// TIA Portal V20 export
FUNCTION_BLOCK "Sequence_2_VisionController"   // FB121, LAD
TITLE = Sequence
// Sequence template programmend in ladder logic
// stored: IsIECCheckEnabled true, MemoryReserve 100, Namespace Unit1.Em6, SetENOAutomatically true
   VAR_OUTPUT
      safeState : Bool;
   END_VAR
   VAR
      statSelectedJobNumber { ExternalWritable := 'False'} : DInt;   // Evaluated Job Number
      instSequenceLADControl { ExternalWritable := 'False'} : "LAF_ControlLadSequence";
      instSequenceLADStatus { ExternalWritable := 'False'} : "LAF_StatusLadSequence";
      statResetJobs { ExternalWritable := 'False'} : Bool;
      statPulse { ExternalWritable := 'False'} : Array[0..999] of Bool;
      statTonTimer { ExternalWritable := 'False'} : Array[0..999] of TON_TIME;
   END_VAR
   VAR_TEMP
      tempCustomerAction : Bool;   // Placeholder for possible actions
      tempDo_nothing_and_wait_for_init : Bool;   // Placeholder for doing nothing
      tempSafeStateCondition : Bool;   // Temp Condition for the equipment module to be in a safe state
   END_VAR
   VAR CONSTANT
      STEP_IDLE : DInt := 1;   // Idle Step
      JOB_1_STEP_01 : DInt := 101;   // Template Step
      JOB_1_STEP_11 : DInt := 111;   // Template Step
      JOB_1_STEP_21 : DInt := 121;   // Template Step
      JOB_1_STEP_31 : DInt := 131;   // Template Step
      JOB_1_STEP_91 : DInt := 191;   // Template Step
      JOB_2_STEP_01 : DInt := 201;   // Template Step
      JOB_2_STEP_11 : DInt := 211;   // Template Step
      JOB_2_STEP_21 : DInt := 221;   // Template Step
      JOB_2_STEP_91 : DInt := 291;   // Template Step
      STEP_IMMEDIATE_STOP : DInt := 901;   // Step executed when an immediate stop command is triggered for the sequence (i.e. when unit is in state aborting)
      SeqDelayTime : Time := T#100ms;
      SeqNoDelayTime : Time;
      TRUE : Bool := TRUE;
      FALSE : Bool := FALSE;
   END_VAR
   VAR_TEMP   // added for the SCL form of the ladder/FBD networks
      _w1 : Bool;
   END_VAR
BEGIN

REGION Network 1: BLOCK INFO HEADER
   // (company) / (C) Copyright (year)
   // ---------------------------------------------------------------------------------
   // Title:                             (Title of this block)
   // Comment/Function: (that is implemented in the block)
   // Library/Family:           (that the source is dedicated to)
   // Author:                        (department / person in charge / contact)
   // Target System:          (test system with FW version)
   // Engineering:              TIA Portal (SW version)
   // Restrictions:               (OB types, etc.)
   // Requirements:           (hardware, technological package, etc.)
   // ---------------------------------------------------------------------------------
   // Change log table:
   // Version          | Date             | Signature      | Expert in charge  | Changes applied ------------------------|----------------------|-------------------------|--------------------------------|-----------------------
   // 001.000.000 | yyyy-mm-dd | 0x00000000 | (name of expert) | First released version
END_REGION

REGION Network 2: DESCRIPTION
   // This is a template block provided by the Automation Framework. It can be used to create an own project.
   // The Block Info Header is prepared to put in your own data.
   // Description of the block could be added here and the docu created by Code2Docu.
END_REGION

REGION Network 3: ******************** CONTROL ********************
END_REGION

REGION Network 4: Sequence Control
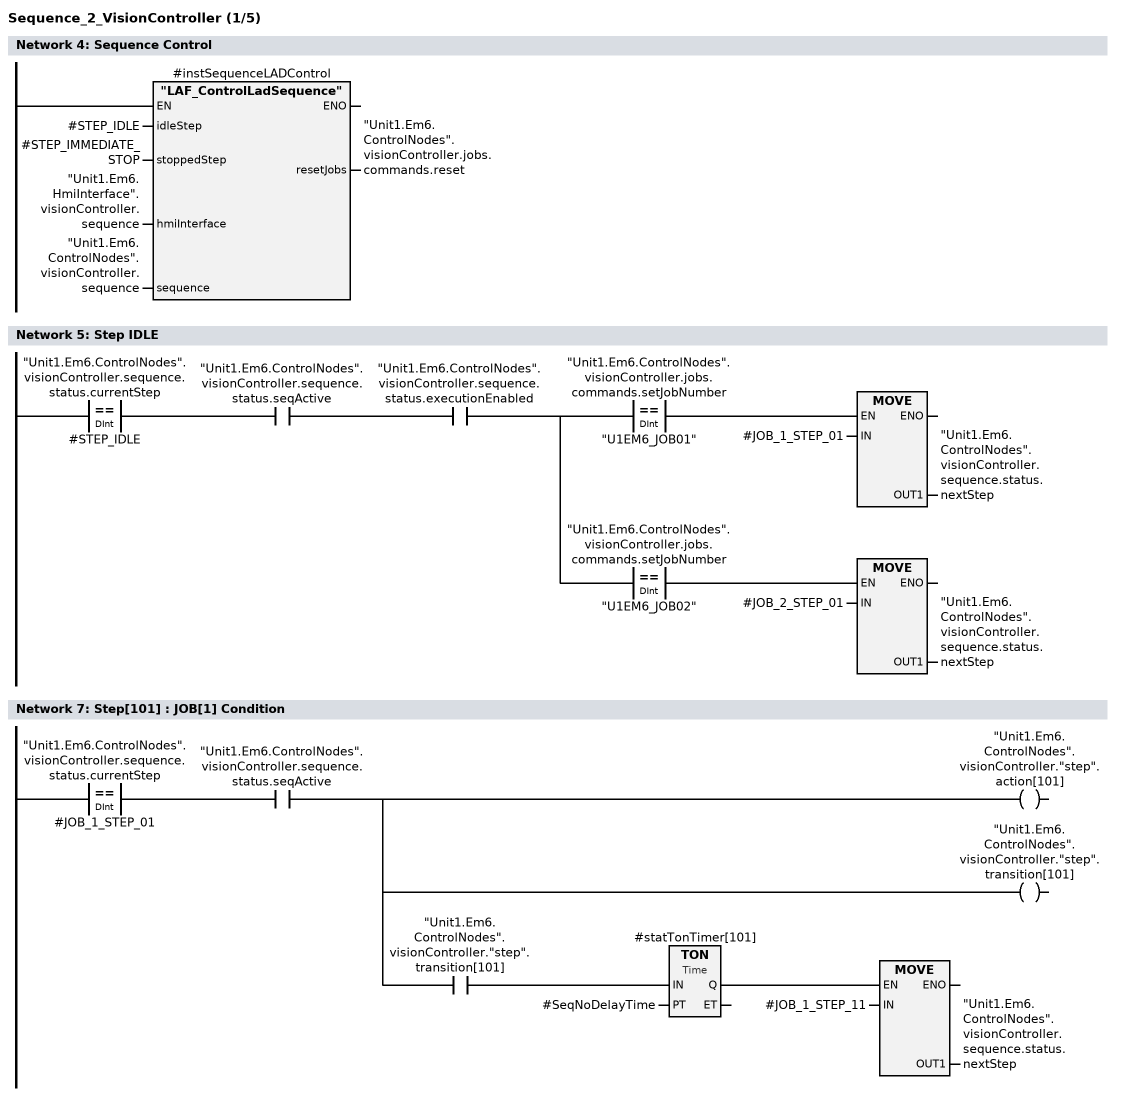
   RUNG wire#powerrail
      #instSequenceLADControl(idleStep := #STEP_IDLE, stoppedStep := #STEP_IMMEDIATE_STOP, hmiInterface := "Unit1.Em6.HmiInterface".visionController.sequence, sequence := "Unit1.Em6.ControlNodes".visionController.sequence, resetJobs => "Unit1.Em6.ControlNodes".visionController.jobs.commands.reset)
   END_RUNG
   // the same network as SCL:
   #instSequenceLADControl(idleStep := #STEP_IDLE,   // "LAF_ControlLadSequence"
                           stoppedStep := #STEP_IMMEDIATE_STOP,
                           hmiInterface := "Unit1.Em6.HmiInterface".visionController.sequence,
                           sequence := "Unit1.Em6.ControlNodes".visionController.sequence,
                           resetJobs => "Unit1.Em6.ControlNodes".visionController.jobs.commands.reset);
END_REGION

REGION Network 5: Step IDLE
   RUNG wire#powerrail
      { S7_Templates := "SrcType := DInt" } EQ_Contact(in1 := "Unit1.Em6.ControlNodes".visionController.sequence.status.currentStep, in2 := #STEP_IDLE)
      Contact( "Unit1.Em6.ControlNodes".visionController.sequence.status.seqActive )
      Contact( "Unit1.Em6.ControlNodes".visionController.sequence.status.executionEnabled )
      wire#w1
      { S7_Templates := "SrcType := DInt" } EQ_Contact(in1 := "Unit1.Em6.ControlNodes".visionController.jobs.commands.setJobNumber, in2 := "U1EM6_JOB01")
      Move(in := #JOB_1_STEP_01, out1 => "Unit1.Em6.ControlNodes".visionController.sequence.status.nextStep)
   END_RUNG
   RUNG wire#w1
      { S7_Templates := "SrcType := DInt" } EQ_Contact(in1 := "Unit1.Em6.ControlNodes".visionController.jobs.commands.setJobNumber, in2 := "U1EM6_JOB02")
      Move(in := #JOB_2_STEP_01, out1 => "Unit1.Em6.ControlNodes".visionController.sequence.status.nextStep)
   END_RUNG
   // the same network as SCL:
   #_w1 := ("Unit1.Em6.ControlNodes".visionController.sequence.status.currentStep = #STEP_IDLE) AND "Unit1.Em6.ControlNodes".visionController.sequence.status.seqActive AND "Unit1.Em6.ControlNodes".visionController.sequence.status.executionEnabled;
   IF #_w1 AND ("Unit1.Em6.ControlNodes".visionController.jobs.commands.setJobNumber = "U1EM6_JOB01") THEN
       "Unit1.Em6.ControlNodes".visionController.sequence.status.nextStep := #JOB_1_STEP_01;
   END_IF;
   IF #_w1 AND ("Unit1.Em6.ControlNodes".visionController.jobs.commands.setJobNumber = "U1EM6_JOB02") THEN
       "Unit1.Em6.ControlNodes".visionController.sequence.status.nextStep := #JOB_2_STEP_01;
   END_IF;
END_REGION

REGION Network 6: ******************** JOB[1] EM INITIALIZED ********************
END_REGION

REGION Network 7: Step[101] : JOB[1] Condition
   RUNG wire#powerrail
      { S7_Templates := "SrcType := DInt" } EQ_Contact(in1 := "Unit1.Em6.ControlNodes".visionController.sequence.status.currentStep, in2 := #JOB_1_STEP_01)
      Contact( "Unit1.Em6.ControlNodes".visionController.sequence.status.seqActive )
      wire#w1
      Coil( "Unit1.Em6.ControlNodes".visionController."step".action[101] )
   END_RUNG
   RUNG wire#w1
      Coil( "Unit1.Em6.ControlNodes".visionController."step".transition[101] )
   END_RUNG
   RUNG wire#w1
      Contact( "Unit1.Em6.ControlNodes".visionController."step".transition[101] )
      { S7_Templates := "time_type := Time" } #statTonTimer[101].TON(pt := #SeqNoDelayTime, et =>)
      Move(in := #JOB_1_STEP_11, out1 => "Unit1.Em6.ControlNodes".visionController.sequence.status.nextStep)
   END_RUNG
   // the same network as SCL:
   "Unit1.Em6.ControlNodes".visionController."step".action[101] := ("Unit1.Em6.ControlNodes".visionController.sequence.status.currentStep = #JOB_1_STEP_01) AND "Unit1.Em6.ControlNodes".visionController.sequence.status.seqActive;
   "Unit1.Em6.ControlNodes".visionController."step".transition[101] := ("Unit1.Em6.ControlNodes".visionController.sequence.status.currentStep = #JOB_1_STEP_01) AND "Unit1.Em6.ControlNodes".visionController.sequence.status.seqActive;
   #statTonTimer[101].TON(IN := ("Unit1.Em6.ControlNodes".visionController.sequence.status.currentStep = #JOB_1_STEP_01) AND "Unit1.Em6.ControlNodes".visionController.sequence.status.seqActive AND "Unit1.Em6.ControlNodes".visionController."step".transition[101],
                          PT := #SeqNoDelayTime);
   IF #statTonTimer[101].Q THEN
       "Unit1.Em6.ControlNodes".visionController.sequence.status.nextStep := #JOB_1_STEP_11;
   END_IF;
END_REGION

REGION Network 8: Step[111] : Vision Controller Ready Check
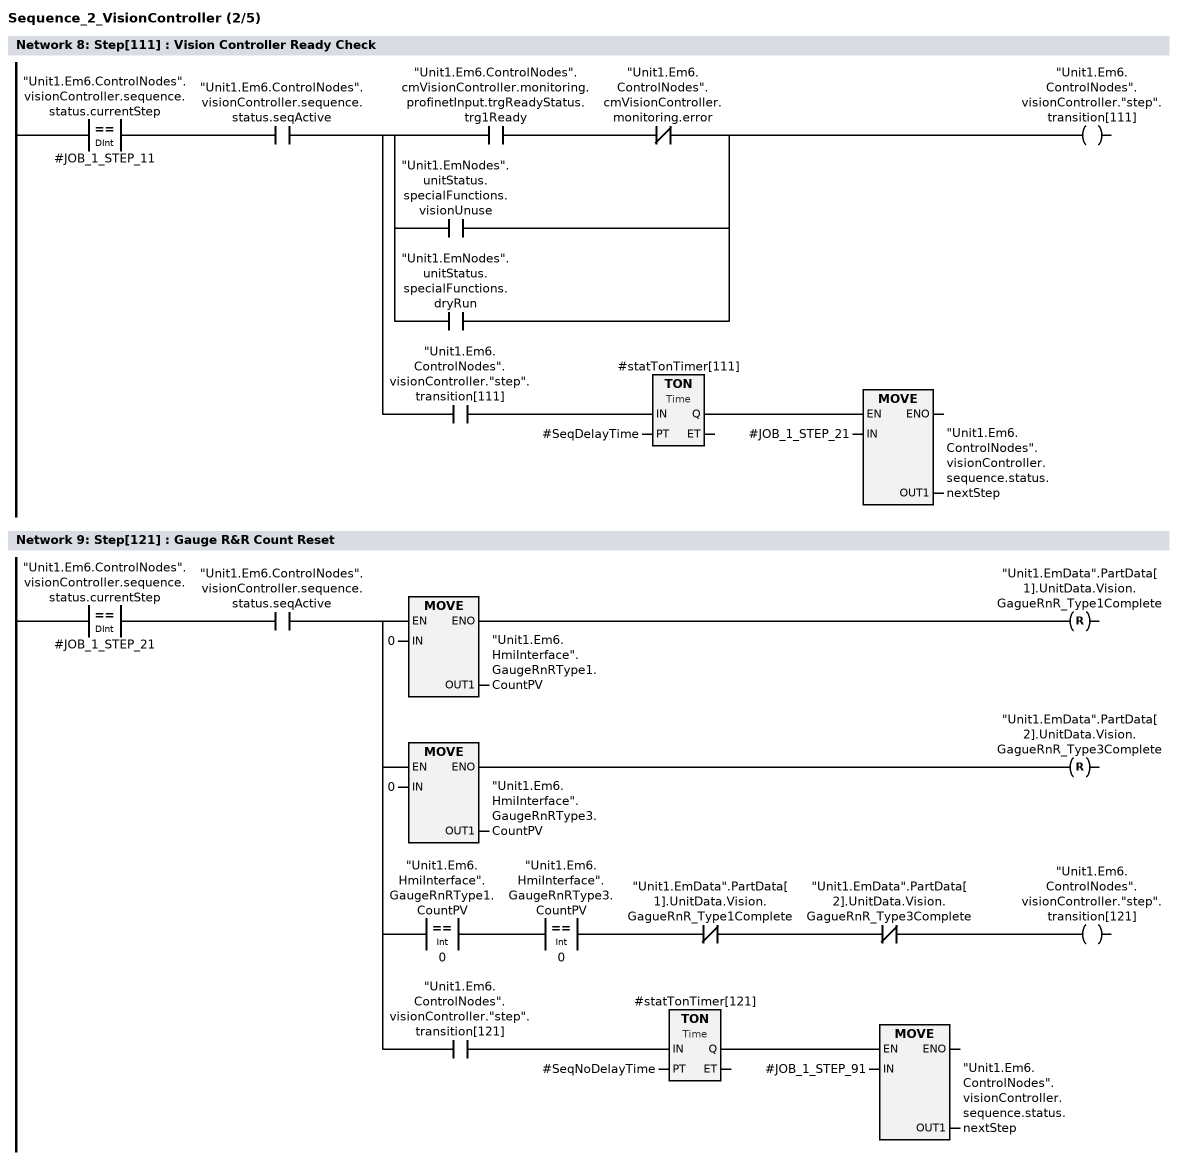
   RUNG wire#powerrail
      { S7_Templates := "SrcType := DInt" } EQ_Contact(in1 := "Unit1.Em6.ControlNodes".visionController.sequence.status.currentStep, in2 := #JOB_1_STEP_11)
      Contact( "Unit1.Em6.ControlNodes".visionController.sequence.status.seqActive )
      wire#w1
      Contact( "Unit1.Em6.ControlNodes".cmVisionController.monitoring.profinetInput.trgReadyStatus.trg1Ready )
      I_Contact( "Unit1.Em6.ControlNodes".cmVisionController.monitoring.error )
      wire#w2
      Coil( "Unit1.Em6.ControlNodes".visionController."step".transition[111] )
   END_RUNG
   RUNG wire#w1
      Contact( "Unit1.EmNodes".unitStatus.specialFunctions.visionUnuse )
   END_RUNG wire#w2
   RUNG wire#w1
      Contact( "Unit1.EmNodes".unitStatus.specialFunctions.dryRun )
   END_RUNG wire#w2
   RUNG wire#w1
      Contact( "Unit1.Em6.ControlNodes".visionController."step".transition[111] )
      { S7_Templates := "time_type := Time" } #statTonTimer[111].TON(pt := #SeqDelayTime, et =>)
      Move(in := #JOB_1_STEP_21, out1 => "Unit1.Em6.ControlNodes".visionController.sequence.status.nextStep)
   END_RUNG
   // the same network as SCL:
   #_w1 := ("Unit1.Em6.ControlNodes".visionController.sequence.status.currentStep = #JOB_1_STEP_11) AND "Unit1.Em6.ControlNodes".visionController.sequence.status.seqActive;
   "Unit1.Em6.ControlNodes".visionController."step".transition[111] := #_w1 AND (("Unit1.Em6.ControlNodes".cmVisionController.monitoring.profinetInput.trgReadyStatus.trg1Ready AND NOT "Unit1.Em6.ControlNodes".cmVisionController.monitoring.error) OR "Unit1.EmNodes".unitStatus.specialFunctions.visionUnuse OR "Unit1.EmNodes".unitStatus.specialFunctions.dryRun);
   #statTonTimer[111].TON(IN := #_w1 AND "Unit1.Em6.ControlNodes".visionController."step".transition[111],
                          PT := #SeqDelayTime);
   IF #statTonTimer[111].Q THEN
       "Unit1.Em6.ControlNodes".visionController.sequence.status.nextStep := #JOB_1_STEP_21;
   END_IF;
END_REGION

REGION Network 9: Step[121] : Gauge R&R Count Reset
   RUNG wire#powerrail
      { S7_Templates := "SrcType := DInt" } EQ_Contact(in1 := "Unit1.Em6.ControlNodes".visionController.sequence.status.currentStep, in2 := #JOB_1_STEP_21)
      Contact( "Unit1.Em6.ControlNodes".visionController.sequence.status.seqActive )
      wire#w1
      Move(in := 0, out1 => "Unit1.Em6.HmiInterface".GaugeRnRType1.CountPV)
      R_Coil( "Unit1.EmData".PartData[1].UnitData.Vision.GagueRnR_Type1Complete )
   END_RUNG
   RUNG wire#w1
      Move(in := 0, out1 => "Unit1.Em6.HmiInterface".GaugeRnRType3.CountPV)
      R_Coil( "Unit1.EmData".PartData[2].UnitData.Vision.GagueRnR_Type3Complete )
   END_RUNG
   RUNG wire#w1
      { S7_Templates := "SrcType := Int" } EQ_Contact(in1 := "Unit1.Em6.HmiInterface".GaugeRnRType1.CountPV, in2 := 0)
      { S7_Templates := "SrcType := Int" } EQ_Contact(in1 := "Unit1.Em6.HmiInterface".GaugeRnRType3.CountPV, in2 := 0)
      I_Contact( "Unit1.EmData".PartData[1].UnitData.Vision.GagueRnR_Type1Complete )
      I_Contact( "Unit1.EmData".PartData[2].UnitData.Vision.GagueRnR_Type3Complete )
      Coil( "Unit1.Em6.ControlNodes".visionController."step".transition[121] )
   END_RUNG
   RUNG wire#w1
      Contact( "Unit1.Em6.ControlNodes".visionController."step".transition[121] )
      { S7_Templates := "time_type := Time" } #statTonTimer[121].TON(pt := #SeqNoDelayTime, et =>)
      Move(in := #JOB_1_STEP_91, out1 => "Unit1.Em6.ControlNodes".visionController.sequence.status.nextStep)
   END_RUNG
   // the same network as SCL:
   #_w1 := ("Unit1.Em6.ControlNodes".visionController.sequence.status.currentStep = #JOB_1_STEP_21) AND "Unit1.Em6.ControlNodes".visionController.sequence.status.seqActive;
   IF #_w1 THEN
       "Unit1.Em6.HmiInterface".GaugeRnRType1.CountPV := 0;
       "Unit1.EmData".PartData[1].UnitData.Vision.GagueRnR_Type1Complete := FALSE;
       "Unit1.Em6.HmiInterface".GaugeRnRType3.CountPV := 0;
       "Unit1.EmData".PartData[2].UnitData.Vision.GagueRnR_Type3Complete := FALSE;
   END_IF;
   "Unit1.Em6.ControlNodes".visionController."step".transition[121] := #_w1 AND ("Unit1.Em6.HmiInterface".GaugeRnRType1.CountPV = 0) AND ("Unit1.Em6.HmiInterface".GaugeRnRType3.CountPV = 0) AND NOT "Unit1.EmData".PartData[1].UnitData.Vision.GagueRnR_Type1Complete AND NOT "Unit1.EmData".PartData[2].UnitData.Vision.GagueRnR_Type3Complete;
   #statTonTimer[121].TON(IN := #_w1 AND "Unit1.Em6.ControlNodes".visionController."step".transition[121],
                          PT := #SeqNoDelayTime);
   IF #statTonTimer[121].Q THEN
       "Unit1.Em6.ControlNodes".visionController.sequence.status.nextStep := #JOB_1_STEP_91;
   END_IF;
END_REGION

REGION Network 10: Step[191] : JOB[1] Step End
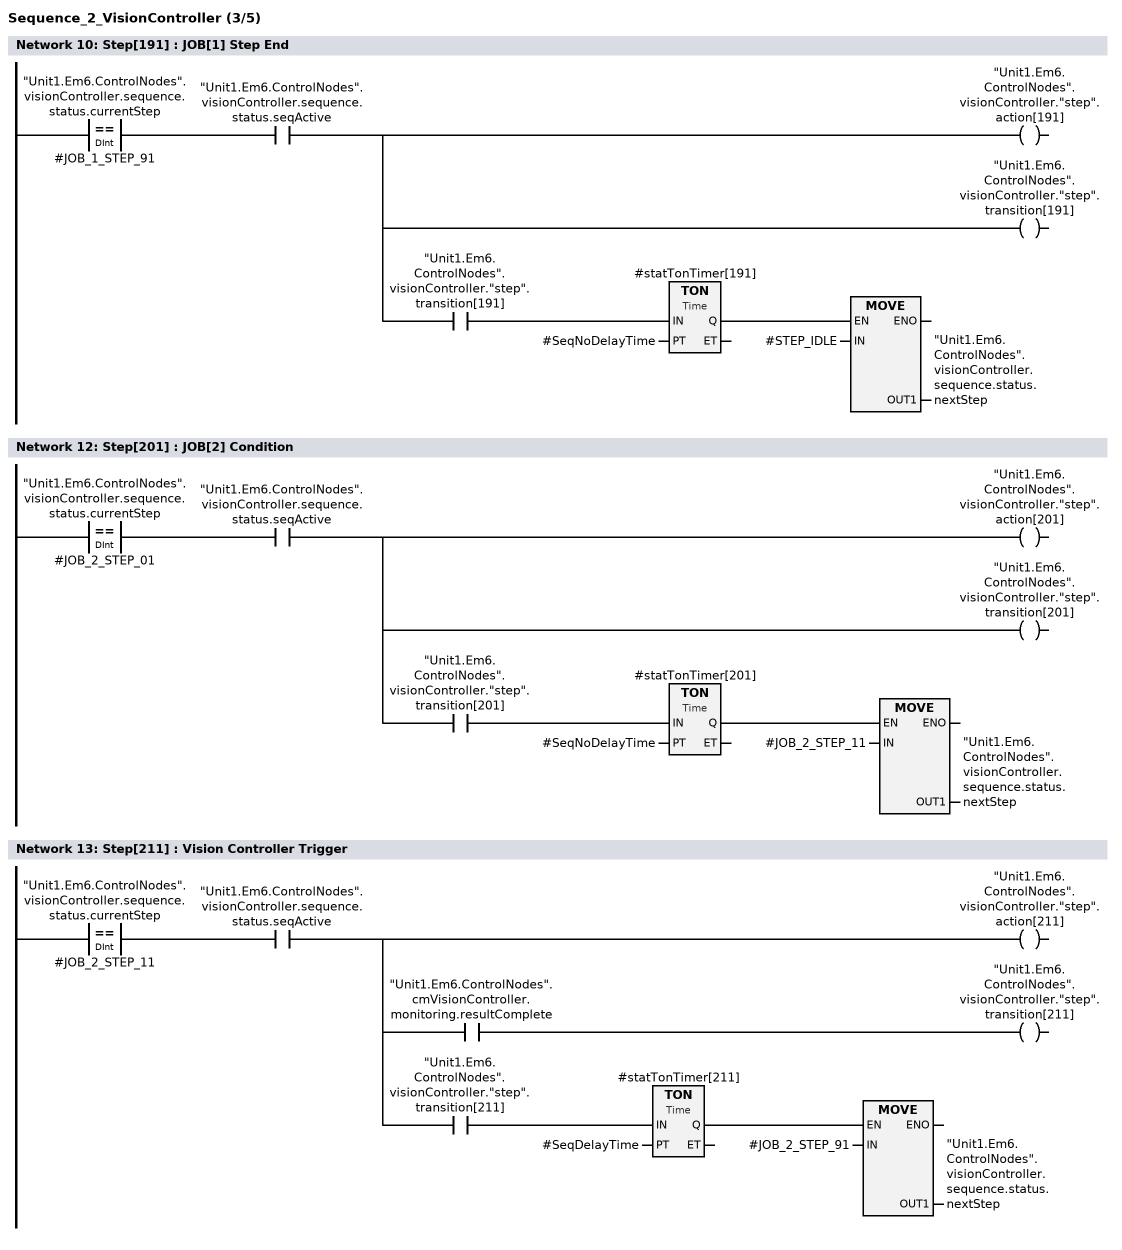
   RUNG wire#powerrail
      { S7_Templates := "SrcType := DInt" } EQ_Contact(in1 := "Unit1.Em6.ControlNodes".visionController.sequence.status.currentStep, in2 := #JOB_1_STEP_91)
      Contact( "Unit1.Em6.ControlNodes".visionController.sequence.status.seqActive )
      wire#w1
      Coil( "Unit1.Em6.ControlNodes".visionController."step".action[191] )
   END_RUNG
   RUNG wire#w1
      Coil( "Unit1.Em6.ControlNodes".visionController."step".transition[191] )
   END_RUNG
   RUNG wire#w1
      Contact( "Unit1.Em6.ControlNodes".visionController."step".transition[191] )
      { S7_Templates := "time_type := Time" } #statTonTimer[191].TON(pt := #SeqNoDelayTime, et =>)
      Move(in := #STEP_IDLE, out1 => "Unit1.Em6.ControlNodes".visionController.sequence.status.nextStep)
   END_RUNG
   // the same network as SCL:
   "Unit1.Em6.ControlNodes".visionController."step".action[191] := ("Unit1.Em6.ControlNodes".visionController.sequence.status.currentStep = #JOB_1_STEP_91) AND "Unit1.Em6.ControlNodes".visionController.sequence.status.seqActive;
   "Unit1.Em6.ControlNodes".visionController."step".transition[191] := ("Unit1.Em6.ControlNodes".visionController.sequence.status.currentStep = #JOB_1_STEP_91) AND "Unit1.Em6.ControlNodes".visionController.sequence.status.seqActive;
   #statTonTimer[191].TON(IN := ("Unit1.Em6.ControlNodes".visionController.sequence.status.currentStep = #JOB_1_STEP_91) AND "Unit1.Em6.ControlNodes".visionController.sequence.status.seqActive AND "Unit1.Em6.ControlNodes".visionController."step".transition[191],
                          PT := #SeqNoDelayTime);
   IF #statTonTimer[191].Q THEN
       "Unit1.Em6.ControlNodes".visionController.sequence.status.nextStep := #STEP_IDLE;
   END_IF;
END_REGION

REGION Network 11: ******************** JOB[2] VISION UNIT INSPECTION AUTO ********************
END_REGION

REGION Network 12: Step[201] : JOB[2] Condition
   RUNG wire#powerrail
      { S7_Templates := "SrcType := DInt" } EQ_Contact(in1 := "Unit1.Em6.ControlNodes".visionController.sequence.status.currentStep, in2 := #JOB_2_STEP_01)
      Contact( "Unit1.Em6.ControlNodes".visionController.sequence.status.seqActive )
      wire#w1
      Coil( "Unit1.Em6.ControlNodes".visionController."step".action[201] )
   END_RUNG
   RUNG wire#w1
      Coil( "Unit1.Em6.ControlNodes".visionController."step".transition[201] )
   END_RUNG
   RUNG wire#w1
      Contact( "Unit1.Em6.ControlNodes".visionController."step".transition[201] )
      { S7_Templates := "time_type := Time" } #statTonTimer[201].TON(pt := #SeqNoDelayTime, et =>)
      Move(in := #JOB_2_STEP_11, out1 => "Unit1.Em6.ControlNodes".visionController.sequence.status.nextStep)
   END_RUNG
   // the same network as SCL:
   "Unit1.Em6.ControlNodes".visionController."step".action[201] := ("Unit1.Em6.ControlNodes".visionController.sequence.status.currentStep = #JOB_2_STEP_01) AND "Unit1.Em6.ControlNodes".visionController.sequence.status.seqActive;
   "Unit1.Em6.ControlNodes".visionController."step".transition[201] := ("Unit1.Em6.ControlNodes".visionController.sequence.status.currentStep = #JOB_2_STEP_01) AND "Unit1.Em6.ControlNodes".visionController.sequence.status.seqActive;
   #statTonTimer[201].TON(IN := ("Unit1.Em6.ControlNodes".visionController.sequence.status.currentStep = #JOB_2_STEP_01) AND "Unit1.Em6.ControlNodes".visionController.sequence.status.seqActive AND "Unit1.Em6.ControlNodes".visionController."step".transition[201],
                          PT := #SeqNoDelayTime);
   IF #statTonTimer[201].Q THEN
       "Unit1.Em6.ControlNodes".visionController.sequence.status.nextStep := #JOB_2_STEP_11;
   END_IF;
END_REGION

REGION Network 13: Step[211] : Vision Controller Trigger
   RUNG wire#powerrail
      { S7_Templates := "SrcType := DInt" } EQ_Contact(in1 := "Unit1.Em6.ControlNodes".visionController.sequence.status.currentStep, in2 := #JOB_2_STEP_11)
      Contact( "Unit1.Em6.ControlNodes".visionController.sequence.status.seqActive )
      wire#w1
      Coil( "Unit1.Em6.ControlNodes".visionController."step".action[211] )
   END_RUNG
   RUNG wire#w1
      Contact( "Unit1.Em6.ControlNodes".cmVisionController.monitoring.resultComplete )
      Coil( "Unit1.Em6.ControlNodes".visionController."step".transition[211] )
   END_RUNG
   RUNG wire#w1
      Contact( "Unit1.Em6.ControlNodes".visionController."step".transition[211] )
      { S7_Templates := "time_type := Time" } #statTonTimer[211].TON(pt := #SeqDelayTime, et =>)
      Move(in := #JOB_2_STEP_91, out1 => "Unit1.Em6.ControlNodes".visionController.sequence.status.nextStep)
   END_RUNG
   // the same network as SCL:
   "Unit1.Em6.ControlNodes".visionController."step".action[211] := ("Unit1.Em6.ControlNodes".visionController.sequence.status.currentStep = #JOB_2_STEP_11) AND "Unit1.Em6.ControlNodes".visionController.sequence.status.seqActive;
   "Unit1.Em6.ControlNodes".visionController."step".transition[211] := ("Unit1.Em6.ControlNodes".visionController.sequence.status.currentStep = #JOB_2_STEP_11) AND "Unit1.Em6.ControlNodes".visionController.sequence.status.seqActive AND "Unit1.Em6.ControlNodes".cmVisionController.monitoring.resultComplete;
   #statTonTimer[211].TON(IN := ("Unit1.Em6.ControlNodes".visionController.sequence.status.currentStep = #JOB_2_STEP_11) AND "Unit1.Em6.ControlNodes".visionController.sequence.status.seqActive AND "Unit1.Em6.ControlNodes".visionController."step".transition[211],
                          PT := #SeqDelayTime);
   IF #statTonTimer[211].Q THEN
       "Unit1.Em6.ControlNodes".visionController.sequence.status.nextStep := #JOB_2_STEP_91;
   END_IF;
END_REGION

REGION Network 14: Step[291] : JOB[2] Step End
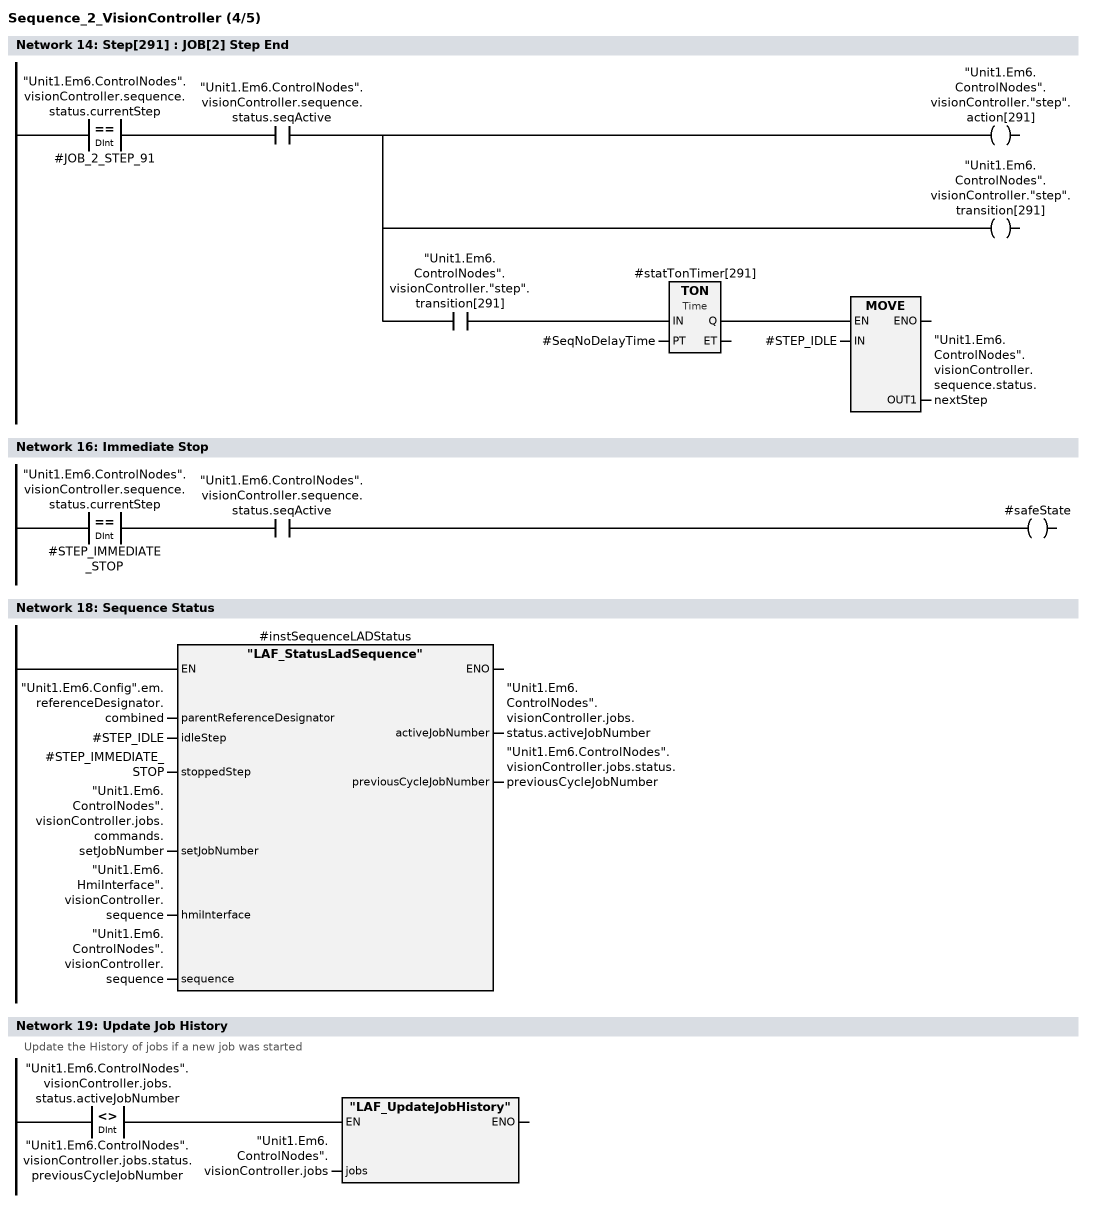
   RUNG wire#powerrail
      { S7_Templates := "SrcType := DInt" } EQ_Contact(in1 := "Unit1.Em6.ControlNodes".visionController.sequence.status.currentStep, in2 := #JOB_2_STEP_91)
      Contact( "Unit1.Em6.ControlNodes".visionController.sequence.status.seqActive )
      wire#w1
      Coil( "Unit1.Em6.ControlNodes".visionController."step".action[291] )
   END_RUNG
   RUNG wire#w1
      Coil( "Unit1.Em6.ControlNodes".visionController."step".transition[291] )
   END_RUNG
   RUNG wire#w1
      Contact( "Unit1.Em6.ControlNodes".visionController."step".transition[291] )
      { S7_Templates := "time_type := Time" } #statTonTimer[291].TON(pt := #SeqNoDelayTime, et =>)
      Move(in := #STEP_IDLE, out1 => "Unit1.Em6.ControlNodes".visionController.sequence.status.nextStep)
   END_RUNG
   // the same network as SCL:
   "Unit1.Em6.ControlNodes".visionController."step".action[291] := ("Unit1.Em6.ControlNodes".visionController.sequence.status.currentStep = #JOB_2_STEP_91) AND "Unit1.Em6.ControlNodes".visionController.sequence.status.seqActive;
   "Unit1.Em6.ControlNodes".visionController."step".transition[291] := ("Unit1.Em6.ControlNodes".visionController.sequence.status.currentStep = #JOB_2_STEP_91) AND "Unit1.Em6.ControlNodes".visionController.sequence.status.seqActive;
   #statTonTimer[291].TON(IN := ("Unit1.Em6.ControlNodes".visionController.sequence.status.currentStep = #JOB_2_STEP_91) AND "Unit1.Em6.ControlNodes".visionController.sequence.status.seqActive AND "Unit1.Em6.ControlNodes".visionController."step".transition[291],
                          PT := #SeqNoDelayTime);
   IF #statTonTimer[291].Q THEN
       "Unit1.Em6.ControlNodes".visionController.sequence.status.nextStep := #STEP_IDLE;
   END_IF;
END_REGION

REGION Network 15: *************** IMMEDIATE STOP ****************
END_REGION

REGION Network 16: Immediate Stop
   RUNG wire#powerrail
      { S7_Templates := "SrcType := DInt" } EQ_Contact(in1 := "Unit1.Em6.ControlNodes".visionController.sequence.status.currentStep, in2 := #STEP_IMMEDIATE_STOP)
      Contact( "Unit1.Em6.ControlNodes".visionController.sequence.status.seqActive )
      Coil( #safeState )
   END_RUNG
   // the same network as SCL:
   #safeState := ("Unit1.Em6.ControlNodes".visionController.sequence.status.currentStep = #STEP_IMMEDIATE_STOP) AND "Unit1.Em6.ControlNodes".visionController.sequence.status.seqActive;
END_REGION

REGION Network 17: *************** STATUS **********************
END_REGION

REGION Network 18: Sequence Status
   RUNG wire#powerrail
      #instSequenceLADStatus(parentReferenceDesignator := "Unit1.Em6.Config".em.referenceDesignator.combined, idleStep := #STEP_IDLE, stoppedStep := #STEP_IMMEDIATE_STOP, setJobNumber := "Unit1.Em6.ControlNodes".visionController.jobs.commands.setJobNumber, hmiInterface := "Unit1.Em6.HmiInterface".visionController.sequence, sequence := "Unit1.Em6.ControlNodes".visionController.sequence, activeJobNumber => "Unit1.Em6.ControlNodes".visionController.jobs.status.activeJobNumber, previousCycleJobNumber => "Unit1.Em6.ControlNodes".visionController.jobs.status.previousCycleJobNumber)
   END_RUNG
   // the same network as SCL:
   #instSequenceLADStatus(parentReferenceDesignator := "Unit1.Em6.Config".em.referenceDesignator.combined,   // "LAF_StatusLadSequence"
                          idleStep := #STEP_IDLE,
                          stoppedStep := #STEP_IMMEDIATE_STOP,
                          setJobNumber := "Unit1.Em6.ControlNodes".visionController.jobs.commands.setJobNumber,
                          hmiInterface := "Unit1.Em6.HmiInterface".visionController.sequence,
                          sequence := "Unit1.Em6.ControlNodes".visionController.sequence,
                          activeJobNumber => "Unit1.Em6.ControlNodes".visionController.jobs.status.activeJobNumber,
                          previousCycleJobNumber => "Unit1.Em6.ControlNodes".visionController.jobs.status.previousCycleJobNumber);
END_REGION

REGION Network 19: Update Job History
   // Update the History of jobs if a new job was started
   RUNG wire#powerrail
      { S7_Templates := "SrcType := DInt" } NE_Contact(in1 := "Unit1.Em6.ControlNodes".visionController.jobs.status.activeJobNumber, in2 := "Unit1.Em6.ControlNodes".visionController.jobs.status.previousCycleJobNumber)
      "LAF_UpdateJobHistory"(jobs := "Unit1.Em6.ControlNodes".visionController.jobs)
   END_RUNG
   // the same network as SCL:
   IF "Unit1.Em6.ControlNodes".visionController.jobs.status.activeJobNumber <> "Unit1.Em6.ControlNodes".visionController.jobs.status.previousCycleJobNumber THEN
       "LAF_UpdateJobHistory"(jobs := "Unit1.Em6.ControlNodes".visionController.jobs);
   END_IF;
END_REGION

REGION Network 20: Output steps as String
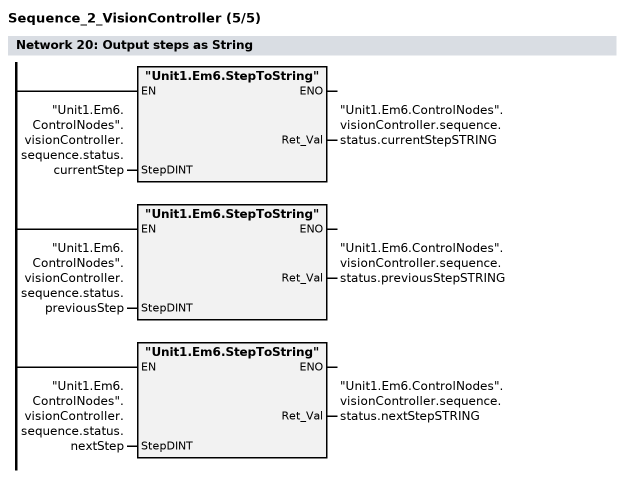
   RUNG wire#powerrail
      "Unit1.Em6.StepToString"(StepDINT := "Unit1.Em6.ControlNodes".visionController.sequence.status.currentStep, Ret_Val => "Unit1.Em6.ControlNodes".visionController.sequence.status.currentStepSTRING)
   END_RUNG
   RUNG wire#powerrail
      "Unit1.Em6.StepToString"(StepDINT := "Unit1.Em6.ControlNodes".visionController.sequence.status.previousStep, Ret_Val => "Unit1.Em6.ControlNodes".visionController.sequence.status.previousStepSTRING)
   END_RUNG
   RUNG wire#powerrail
      "Unit1.Em6.StepToString"(StepDINT := "Unit1.Em6.ControlNodes".visionController.sequence.status.nextStep, Ret_Val => "Unit1.Em6.ControlNodes".visionController.sequence.status.nextStepSTRING)
   END_RUNG
   // the same network as SCL:
   "Unit1.Em6.ControlNodes".visionController.sequence.status.currentStepSTRING := "Unit1.Em6.StepToString"(StepDINT := "Unit1.Em6.ControlNodes".visionController.sequence.status.currentStep);
   "Unit1.Em6.ControlNodes".visionController.sequence.status.previousStepSTRING := "Unit1.Em6.StepToString"(StepDINT := "Unit1.Em6.ControlNodes".visionController.sequence.status.previousStep);
   "Unit1.Em6.ControlNodes".visionController.sequence.status.nextStepSTRING := "Unit1.Em6.StepToString"(StepDINT := "Unit1.Em6.ControlNodes".visionController.sequence.status.nextStep);
END_REGION
END_FUNCTION_BLOCK
